(* CoDeSys 2.3.9.41 project: revolution.pro *)
(* Libraries: STANDARD.LIB 4.10.05 10:14:46, IECSFC.LIB 13.4.06 14:51:28, SYSLIBTIME.LIB 20.2.06 13:31:16, SYSTASKINFO.LIB 20.2.06 13:31:38, ANALYZATION.LIB 5.10.99 08:05:06, SYSLIBCALLBACK.LIB 20.2.06 13:31:08, PID_Regulators.lib 28.12.06 17:47:54 *)

(* PLC configuration (modules and I/O channels)
DI0_EKM AT %IX0.0 [BitInput]
DI1_pmp1confirm AT %IX0.1 [BitInput]
DI2_pmp2confirm AT %IX0.2 [BitInput]
DI3_pmp3confirm AT %IX0.3 [BitInput]
DI4_pmp1auto AT %IX0.4 [BitInput]
DI5_pmp2auto AT %IX0.5 [BitInput]
Discrete output 4 bit [ID101] node 1, in %IB1 out %QB1 {PinCount = 4; SafeValueBool = FALSE; SafeValueBool = FALSE; SafeValueBool = FALSE; SafeValueBool = FALSE; Visibility = No}
  DO0_pmp1 AT %QX1.0 [BitOutput]
  DO1_pmp2 AT %QX1.1 [BitOutput]
  DO2_pmp3 AT %QX1.2 [BitOutput]
  DO_alarmLight AT %QX1.3 [BitOutput]
Special output [ID104] node 2, in %IB2 out %QB2 {Visibility = No; PinCount = 1}
  AT %QX2.0 [BitOutput] Special output
AI_pressure AT %ID3.0 [FloatInput] Value
cirTime AT %IW3.1 [WordInput] Circular time
Analog Input [ID107] node 0, in %IB3.0 out %QB3.0
Unifed signal sensor [ID700] node 4, in %IB4 out %QB4 {Type_of_sensor700 = IT_0_20; measure_interval = 0.5; ainlow = 0; ainhigh = 20; first_cor_point = 0; first_delta = 0; second_cor_point = 0; second_delta = 0; third_cor_point = 0; third_delta = 0; Visibility = No}
  AT %ID4.0 [FloatInput] Value
  AT %IW4.1 [WordInput] Circular time
  Analog Input [ID107] node 0, in %IB4.0 out %QB4.0
Unifed signal sensor [ID700] node 5, in %IB5 out %QB5 {Type_of_sensor700 = IT_0_20; measure_interval = 0.5; ainlow = 0; ainhigh = 20; first_cor_point = 0; first_delta = 0; second_cor_point = 0; second_delta = 0; third_cor_point = 0; third_delta = 0; Visibility = No}
  AT %ID5.0 [FloatInput] Value
  AT %IW5.1 [WordInput] Circular time
  Analog Input [ID107] node 0, in %IB5.0 out %QB5.0
Unifed signal sensor [ID700] node 6, in %IB6 out %QB6 {Type_of_sensor700 = IT_0_20; measure_interval = 0.5; ainlow = 0; ainhigh = 20; first_cor_point = 0; first_delta = 0; second_cor_point = 0; second_delta = 0; third_cor_point = 0; third_delta = 0; Visibility = No}
  AT %ID6.0 [FloatInput] Value
  AT %IW6.1 [WordInput] Circular time
  Analog Input [ID107] node 0, in %IB6.0 out %QB6.0
Analog output [ID106] node 7, in %IB7 out %QB7 {DAC_Type = Voltage 0-10 B; Analog_offset_correction = 0; Analog_full_range_correction = 0; SafeValueFloat = 0; Visibility = No}
  AT %QD7.0 [FloatOutput] Value
  AT %QD8.0 [FloatOutput] Value
AT %QD9.0 [DWordOutput] Last address
AT %QW9.1 [WordOutput] Last error
RS-485-1 [COM1_USART] node 0, in %IB9.0 out %QB9.0 {CommunicationSpeed = 19200; Parity = NO PARITY CHECK; BitLength = 8 bits; StopLength = One stop bit; InterfaceType = RS485; FrameOriented = RTU; Timeout = 0; Visibility = No}
AT %QB9.1.0 [ComChannel] Command (0xff - Start)
atv1_freq AT %IW9.1.0.0 [WordInput]
atv1_curr AT %IW9.1.1.0 [WordInput]
atv1_lastError AT %IW9.1.2.0 [WordInput]
atv1_writeHz AT %QW9.1.3.0 [WordOutput]
AT %QB9.2.0 [ComChannel] Command (0xff - Start)
atv2_freq AT %IW9.2.0.0 [WordInput]
atv2_curr AT %IW9.2.1.0 [WordInput]
atv2_lastError AT %IW9.2.2.0 [WordInput]
atv2_writeHz AT %QW9.2.3.0 [WordOutput]
Debug RS-232 [DEBUG_USART] node 0, in %IB10.0.0 out %QB10.0.0 {CommunicationSpeed = 11520; Parity = EVEN; BitLength = 8 bits; StopLength = One stop bit; InterfaceType = RS232; FrameOriented = RTU; Timeout = 0; Visibility = No}
pan_INPUT_ONE AT %QW10.1.0 [WordOutput] setTime
pan_INPUT_TWO AT %QW10.2.0 [WordOutput]
pan_OUTPUT_ONE AT %QW10.3.0 [WordOutput]
pan_OUTPUT_TWO AT %QW10.4.0 [WordOutput]
2 byte [Register] node 5, in %IB10.5 out %QB10.5
  pan_pressure AT %QW10.5.0 [WordOutput]
2 byte [Register] node 6, in %IB10.6 out %QB10.6
  pan_daySetpoint AT %QW10.6.0 [WordOutput]
2 byte [Register] node 7, in %IB10.7 out %QB10.7
  pan_nightSetpoint AT %QW10.7.0 [WordOutput]
2 byte [Register] node 8, in %IB10.8 out %QB10.8
  pan_finishSetpoint AT %QW10.8.0 [WordOutput]
2 byte [Register] node 9, in %IB10.9 out %QB10.9
  pan_pres4ma AT %QW10.9.0 [WordOutput]
2 byte [Register] node 10, in %IB10.10 out %QB10.10
  pan_pres20ma AT %QW10.10.0 [WordOutput]
2 byte [Register] node 11, in %IB10.11 out %QB10.11
  pan_mainPmp AT %QW10.11.0 [WordOutput]
2 byte [Register] node 12, in %IB10.12 out %QB10.12
  pan_resStartDelta AT %QW10.12.0 [WordOutput]
2 byte [Register] node 13, in %IB10.13 out %QB10.13
  pan_resStartDelay AT %QW10.13.0 [WordOutput]
2 byte [Register] node 14, in %IB10.14 out %QB10.14
  pan_resStopHz AT %QW10.14.0 [WordOutput]
2 byte [Register] node 15, in %IB10.15 out %QB10.15
  pan_prop AT %QW10.15.0 [WordOutput]
2 byte [Register] node 16, in %IB10.16 out %QB10.16
  pan_integ AT %QW10.16.0 [WordOutput]
2 byte [Register] node 17, in %IB10.17 out %QB10.17
  pan_diff AT %QW10.17.0 [WordOutput]
2 byte [Register] node 18, in %IB10.18 out %QB10.18
  pan_integMin AT %QW10.18.0 [WordOutput]
2 byte [Register] node 19, in %IB10.19 out %QB10.19
  pan_integMax AT %QW10.19.0 [WordOutput]
2 byte [Register] node 20, in %IB10.20 out %QB10.20
  pan_dryHodDelay AT %QW10.20.0 [WordOutput]
2 byte [Register] node 21, in %IB10.21 out %QB10.21
  pan_aType_1 AT %QW10.21.0 [WordOutput]
2 byte [Register] node 22, in %IB10.22 out %QB10.22
  pan_aType_2 AT %QW10.22.0 [WordOutput]
2 byte [Register] node 23, in %IB10.23 out %QB10.23
  pan_aType_3 AT %QW10.23.0 [WordOutput]
2 byte [Register] node 24, in %IB10.24 out %QB10.24
  pan_aTime_1 AT %QW10.24.0 [WordOutput]
2 byte [Register] node 25, in %IB10.25 out %QB10.25
  pan_aTime_2 AT %QW10.25.0 [WordOutput]
2 byte [Register] node 26, in %IB10.26 out %QB10.26
  pan_aTime_3 AT %QW10.26.0 [WordOutput]
2 byte [Register] node 27, in %IB10.27 out %QB10.27
  pan_aDate_1 AT %QW10.27.0 [WordOutput]
2 byte [Register] node 28, in %IB10.28 out %QB10.28
  pan_aDate_2 AT %QW10.28.0 [WordOutput]
2 byte [Register] node 29, in %IB10.29 out %QB10.29
  pan_aDate_3 AT %QW10.29.0 [WordOutput]
2 byte [Register] node 30, in %IB10.30 out %QB10.30
  pan_aPres_1 AT %QW10.30.0 [WordOutput]
2 byte [Register] node 31, in %IB10.31 out %QB10.31
  pan_aPres_2 AT %QW10.31.0 [WordOutput]
2 byte [Register] node 32, in %IB10.32 out %QB10.32
  pan_aPres_3 AT %QW10.32.0 [WordOutput]
2 byte [Register] node 33, in %IB10.33 out %QB10.33
  pan_aSetpoint_1 AT %QW10.33.0 [WordOutput]
2 byte [Register] node 34, in %IB10.34 out %QB10.34
  pan_aSetpoint_2 AT %QW10.34.0 [WordOutput]
2 byte [Register] node 35, in %IB10.35 out %QB10.35
  pan_aSetpoint_3 AT %QW10.35.0 [WordOutput]
2 byte [Register] node 36, in %IB10.36 out %QB10.36
  pan_aFreq_1 AT %QW10.36.0 [WordOutput]
2 byte [Register] node 37, in %IB10.37 out %QB10.37
  pan_aFreq_2 AT %QW10.37.0 [WordOutput]
2 byte [Register] node 38, in %IB10.38 out %QB10.38
  pan_aFreq_3 AT %QW10.38.0 [WordOutput]
2 byte [Register] node 39, in %IB10.39 out %QB10.39
  pan_aCurr_1 AT %QW10.39.0 [WordOutput]
2 byte [Register] node 40, in %IB10.40 out %QB10.40
  pan_aCurr_2 AT %QW10.40.0 [WordOutput]
2 byte [Register] node 41, in %IB10.41 out %QB10.41
  pan_aCurr_3 AT %QW10.41.0 [WordOutput]
2 byte [Register] node 42, in %IB10.42 out %QB10.42
  pan_aMainPmp_1 AT %QW10.42.0 [WordOutput]
2 byte [Register] node 43, in %IB10.43 out %QB10.43
  pan_aMainPmp_2 AT %QW10.43.0 [WordOutput]
2 byte [Register] node 44, in %IB10.44 out %QB10.44
  pan_aMainPmp_3 AT %QW10.44.0 [WordOutput]
2 byte [Register] node 45, in %IB10.45 out %QB10.45
  pan_topPos AT %QW10.45.0 [WordOutput]
2 byte [Register] node 46, in %IB10.46 out %QB10.46
  pan_midPos AT %QW10.46.0 [WordOutput]
2 byte [Register] node 47, in %IB10.47 out %QB10.47
  pan_bottomPos AT %QW10.47.0 [WordOutput]
2 byte [Register] node 48, in %IB10.48 out %QB10.48
  pan_cursor AT %QW10.48.0 [WordOutput]
2 byte [Register] node 49, in %IB10.49 out %QB10.49
  pan_setHH AT %QW10.49.0 [WordOutput]
2 byte [Register] node 50, in %IB10.50 out %QB10.50
  pan_setMMin AT %QW10.50.0 [WordOutput]
2 byte [Register] node 51, in %IB10.51 out %QB10.51
  pan_setDD AT %QW10.51.0 [WordOutput]
2 byte [Register] node 52, in %IB10.52 out %QB10.52
  pan_setMM AT %QW10.52.0 [WordOutput]
2 byte [Register] node 53, in %IB10.53 out %QB10.53
  pan_setYY AT %QW10.53.0 [WordOutput]
2 byte [Register] node 54, in %IB10.54 out %QB10.54
  pan_currHH AT %QW10.54.0 [WordOutput]
2 byte [Register] node 55, in %IB10.55 out %QB10.55
  pan_currMMin AT %QW10.55.0 [WordOutput]
2 byte [Register] node 56, in %IB10.56 out %QB10.56
  pan_currDD AT %QW10.56.0 [WordOutput]
2 byte [Register] node 57, in %IB10.57 out %QB10.57
  pan_currYY AT %QW10.57.0 [WordOutput]
  pan_ppDelay AT %QW10.58.0 [WordOutput]
  pan_ppLimit AT %QW10.59.0 [WordOutput]
  pan_ppFic AT %QW10.60.0 [WordOutput]
  AT %QW10.61.0 [WordOutput]
  AT %QW10.62.0 [WordOutput]
*)

(* Global variable list: Global_Variables *)
VAR_GLOBAL
	(* Times *)
	GetTime: CurTimeEx;
	TimeAndDate: SystemTimeDate;
	Sys_Time: SysTime64;

	(* Alarms *)
	Alarmy : WORD;

	sensBreak : BOOL; (* 1 *)
	sensShort : BOOL; (* 2 *)
	dryHod		 : BOOL; (* 3 *)
	ekmUpper : BOOL; (* 4 *)
	fcAlarm	: BOOL; (* 5 *)
	kaPmp1fc	: BOOL; (* 6 *)
	kaPmp2fc	: BOOL; (* 7 *)
	kaPmp3fc : BOOL; (* 8 *)
	kaKM1		: BOOL; (* 9 *)
	kaPmp1d : BOOL;  (* 10 *)
	kaPmp2d : BOOL;  (* 11 *)
	kaPmp3d : BOOL;  (* 12 *)
END_VAR

(* POU PLC_PRG, ST *)
PROGRAM PLC_PRG
VAR
	scale : CALIBRATION;
	spcheck : SPDAYCYCLE;
	core : PNS_CORE;
	priority : PRIORITIZATION;
	rotate : ROTATION;
	protect : PRESSURE_PROTECT;

	(* dryHod *)
	dryTimer : TON;
	dryHodOk : BOOL;

	(* Alarmes *)
	breakDetect : BOOL;
	breakTimer : TON;

	shortDetect : BOOL;
	shortTimer : TON;

	fcAlarmDetect, fcAlarmFP : BOOL;
	fcAlarmTimer : TON;

	pmp1kaDetect, pmp2kaDetect, pmp3kaDetect : BOOL;
	pmp1kaDetectD, pmp2kaDetectD, pmp3kaDetectD : BOOL;
	pmp1kaTimer, pmp2kaTimer, pmp3kaTimer : TON;
	pmp1kaTimerD, pmp2kaTimerD, pmp3kaTimerD : TON;
	pmp1kaFP, pmp2kaFP, pmp3kaFP,  kmKaFP : BOOL;
	pmp1kaFPD, pmp2kaFPD, pmp3kaFPD,  kmKaFPD : BOOL;
	fc_state, fc_kaDetect : BOOL;
	fcKaTimer : TON;

	(* Times *)
	setTime : BOOL;
END_VAR
VAR RETAIN
	(* dry hod *)
	dryDelay : TIME;

	(* Pressure *)
	daySetpoint, nightSetpoint : REAL;

	(*Calibration *)
	pres4ma, pres20ma : REAL;

	(* Process *)
	resStartDelta : REAL;
	resStartDelay : TIME;
	resStopHz : WORD;

	(* PID *)
	prop : REAL;
	integ : DINT;

	(* Pressure Protect *)
	ppDelay : TIME;
	ppLimit : REAL;
	ppFic : REAL;

END_VAR
dryTimer(IN:= DI0_EKM, PT:=dryDelay, Q=>dryHodOk, ET=> );

Inputs;



Times;
END_PROGRAM
ACTION Alarmes:
(* SENS BREAK *)
IF AI_pressure < 3.8 THEN
	breakDetect := TRUE;
ELSE
	breakDetect := FALSE;
END_IF;

breakTimer(IN:= breakDetect, PT:=T#1s, Q=>sensBreak, ET=> );


(* SENS SHORT *)
IF AI_pressure > 21.0 THEN
	shortDetect := TRUE;
ELSE
	shortDetect := FALSE;
END_IF;

shortTimer(IN:= shortDetect, PT:=T#1s, Q=>sensShort, ET=> );

(* DRY HOD *)
dryHod := dryHodOk;

(* EKM UPPER *)

(* FC ALARM *)
(*
IF DI_fcAlarm AND fc_on = TRUE THEN
	fcAlarmDetect := TRUE;
ELSE
	fcAlarmDetect := FALSE;
END_IF;

fcAlarmTimer(IN:= fcAlarmDetect, PT:=T#10s, Q=>fcAlarm, ET=> );

IF fcAlarm AND fcAlarmFP = FALSE THEN
	fcAlarmFP := TRUE;
	ShiftKtpMainPmp;
END_IF;

IF fcAlarm = FALSE THEN
	fcAlarmFP := FALSE;
END_IF;
*)
(* PMP1 KA *)
	(* FC *)
(*
IF pmp1fc AND pmp1_state = FALSE THEN
	pmp1kaDetect := TRUE;
ELSE
	pmp1kaDetect := FALSE;
END_IF;
	(* Direct *)
IF pmp1d AND pmp1_stateD = FALSE THEN
	pmp1kaDetectD := TRUE;
ELSE
	pmp1kaDetectD := FALSE;
END_IF;
*)
(*
pmp1kaTimer(IN:= pmp1kaDetect, PT:=T#10s, Q=>kaPmp1fc, ET=> );
pmp1kaTimerD(IN:= pmp1kaDetectD, PT:=T#10s, Q=>kaPmp1d, ET=> );
*)
(*
(* FC *)
IF kaPmp1fc AND pmp1kaFP = FALSE THEN
	pmp1kaFP := TRUE;
	pmp1kaSave := TRUE;
	ShiftKtpMainPmp;
END_IF;

IF kaPmp1fc = FALSE THEN
	pmp1kaFP := FALSE;
END_IF;
(* Direct *)
IF kaPmp1d AND pmp1kaFPD = FALSE THEN
	pmp1kaFPD := TRUE;
	pmp1kaSaveD := TRUE;
END_IF;

IF kaPmp1d = FALSE THEN
	pmp1kaFPD := FALSE;
END_IF;
*)
(*
(* PMP2 KA *)
IF pmp2fc AND pmp2_state = FALSE THEN
	pmp2kaDetect := TRUE;
ELSE
	pmp2kaDetect := FALSE;
END_IF;

IF pmp2d AND pmp2_stateD = FALSE THEN
	pmp2kaDetectD := TRUE;
ELSE
	pmp2kaDetectD := FALSE;
END_IF;

pmp2kaTimer(IN:= pmp2kaDetect, PT:=T#10s, Q=>kaPmp2fc, ET=> );
pmp2kaTimerD(IN:= pmp2kaDetectD, PT:=T#10s, Q=>kaPmp2d, ET=> );

IF kaPmp2fc AND pmp2kaFP = FALSE THEN
	pmp2kaFP := TRUE;
	pmp2kaSave := TRUE;
END_IF;

IF kaPmp2fc = FALSE THEN
	pmp2kaFP := FALSE;
END_IF;

IF kaPmp2d AND pmp2kaFPD = FALSE THEN
	pmp2kaFPD := TRUE;
	pmp2kaSaveD := TRUE;
END_IF;

IF kaPmp2d = FALSE THEN
	pmp2kaFPD := FALSE;
END_IF;

(* PMP3 KA *)
IF pmp3fc AND pmp3_state = FALSE THEN
	pmp3kaDetect := TRUE;
ELSE
	pmp3kaDetect := FALSE;
END_IF;

IF pmp3d AND pmp3_stateD = FALSE THEN
	pmp3kaDetectD := TRUE;
ELSE
	pmp3kaDetectD := FALSE;
END_IF;

pmp3kaTimer(IN:= pmp3kaDetect, PT:=T#10s, Q=>kaPmp3fc, ET=> );
pmp3kaTimerD(IN:= pmp3kaDetectD, PT:=T#10s, Q=>kaPmp3d, ET=> );

IF kaPmp3fc AND pmp3kaFP = FALSE THEN
	pmp3kaFP := TRUE;
	pmp3kaSave := TRUE;
	ShiftKtpMainPmp;
END_IF;

IF kaPmp3fc = FALSE THEN
	pmp3kaFP := FALSE;
END_IF;

IF kaPmp3d AND pmp3kaFPD = FALSE THEN
	pmp3kaFPD := TRUE;
	pmp3kaSaveD := TRUE;
END_IF;

IF kaPmp3d = FALSE THEN
	pmp3kaFPD := FALSE;
END_IF;

IF ktp_INPUT.1 THEN
	pmp1kaSave := FALSE;
	pmp2kaSave := FALSE;
	pmp3kaSave := FALSE;
	pmp1kaSaveD := FALSE;
	pmp2kaSaveD := FALSE;
	pmp3kaSaveD := FALSE;
	ktp_INPUT.1 := FALSE;
END_IF;

(* FC KA *)
IF fc_on AND fc_state = FALSE THEN
	fc_kaDetect := TRUE;
ELSE
	fc_kaDetect := FALSE;
END_IF;

fcKaTimer(IN:= fc_kaDetect, PT:=T#10s, Q=>kaKM1, ET=> );

IF kaKM1 AND kmKaFP = FALSE THEN
	kmKaFP := TRUE;
	ShiftKtpMainPmp;
END_IF;

IF kaKM1 = FALSE THEN
	kmKaFP := FALSE;
END_IF;

(* ALARMY *)
Alarmy.0 := sensBreak;
Alarmy.1 := sensShort;
Alarmy.2 := dryHod;

Alarmy.4 := fcAlarm;
Alarmy.5 := kaPmp1fc;
Alarmy.6 := kaPmp2fc;
Alarmy.7 := kaPmp3fc;
Alarmy.8 := kaKM1;

IF Alarmy > 0 THEN
	DO_lamp_fcAlarm := TRUE;
ELSE
	DO_lamp_fcAlarm := FALSE;
END_IF;
*)
END_ACTION
ACTION Inputs:
setTime := pan_INPUT_ONE.0;

drydelay := WORD_TO_TIME ( pan_dryHoddelay * 1000 );

daySetpoint := WORD_TO_REAL ( pan_daySetpoint ) / 100;
nightSetpoint := WORD_TO_REAL ( pan_nightSetpoint ) / 100;

pres4ma := WORD_TO_REAL ( pan_pres4ma ) / 100;
pres20ma := WORD_TO_REAL ( pan_pres20ma ) / 100;

resStartDelta := WORD_TO_REAL ( pan_resStartDelta ) / 100;
resStartDelay := WORD_TO_TIME ( pan_resStartDelay * 1000 );
resStopHz := resStopHz;

prop := WORD_TO_REAL ( pan_prop ) / 100;
integ := pan_integ;

ppDelay := WORD_TO_TIME ( pan_ppDelay * 1000 );
ppLimit := WORD_TO_REAL ( pan_ppLimit ) / 100;
ppFic := WORD_TO_REAL ( pan_ppFic ) / 100;
END_ACTION
ACTION Times:
TimeAndDate.Day :=0;
TimeAndDate.DayOfWeek :=0;
TimeAndDate.dwHighMsec :=0;
TimeAndDate.dwLowMSecs :=0;
TimeAndDate.Milliseconds :=0;
TimeAndDate.Minute :=0;
TimeAndDate.Second :=0;
TimeAndDate.Hour :=0;
TimeAndDate.Year :=0;
TimeAndDate.Month :=0;
Sys_time.ulHigh :=0;
Sys_time.ulLow :=0;
GetTime (SystemTime:=Sys_Time , TimeDate:= TimeAndDate);


IF pan_INPUT_ONE.0 THEN
	TimeAndDate.Minute:=pan_setMMin;
	TimeAndDate.Second:=10;
	TimeAndDate.Hour:=pan_setHH;
	TimeAndDate.Day:=pan_setDD;
	TimeAndDate.Month:=pan_setMM;
	TimeAndDate.Year:=pan_setYY;
	GetTime (SystemTime:=Sys_Time , TimeDate:= TimeAndDate);

	pan_INPUT_ONE.0 := FALSE;
END_IF;
END_ACTION

(* POU CALIBRATION, ST *)
FUNCTION_BLOCK CALIBRATION
VAR_INPUT
	AI_RAW : REAL;
	r_bar4ma : REAL;
	w2d_bar4ma : WORD;
	r_bar20ma : REAL;
	w2d_bar20ma : WORD;
END_VAR
VAR_OUTPUT
	r_scaled : REAL;
	w2d_scaled : WORD;
END_VAR
VAR
END_VAR
(* Result = n2 + ( Input - n1 ) * ( ( m2 - n2 ) / ( m1 - n1 ) ) *)

w2d_scaled := w2d_bar4ma  + ( REAL_TO_INT( AI_RAW * 100 ) - 400 ) * ( w2d_bar20ma - w2d_bar4ma ) / 1600;

r_scaled := r_bar4ma  + ( AI_RAW - 4.0 ) * ( r_bar20ma - r_bar4ma ) / 16;
END_FUNCTION_BLOCK

(* POU SPDAYCYCLE, ST *)
FUNCTION_BLOCK SPDAYCYCLE
VAR_INPUT
	firstSetpoint : REAL;
	secondSetpoint : REAL;
	spHHfirst : WORD;
	spMMfirst : WORD;
	spHHsecond : WORD;
	spMMsecond : WORD;
	HH, MM : WORD;
END_VAR
VAR_OUTPUT
	setpoint : REAL;
END_VAR
VAR
END_VAR
IF spHHsecond > spHHfirst THEN
	IF HH = spHHsecond AND MM >= spMMsecond THEN
		setpoint := secondSetpoint;
	END_IF;
	IF HH > spHHsecond AND HH > spHHfirst THEN
		setpoint := secondSetpoint;
	END_IF;
	IF HH >= 0 AND HH < spHHfirst THEN
		setpoint := secondSetpoint;
	END_IF;
	IF HH = spHHfirst AND MM < spMMfirst THEN
		setpoint := secondSetpoint;
	END_IF;
	IF HH = spHHfirst AND MM >= spMMfirst THEN
		setpoint := firstSetpoint;
	END_IF;
	IF HH > spHHfirst AND HH < spHHsecond THEN
		setpoint := firstSetpoint;
	END_IF;
	IF HH = spHHsecond AND MM < spMMsecond THEN
		setpoint := firstSetpoint;
	END_IF;
END_IF;

IF spHHsecond < spHHfirst THEN
	IF HH = spHHsecond AND MM >= spMMsecond THEN
		setpoint := secondSetpoint;
	END_IF;
	IF HH > spHHsecond AND HH < spHHfirst THEN
		setpoint := secondSetpoint;
	END_IF;
	IF HH = spHHfirst AND MM < spMMfirst THEN
		setpoint := secondSetpoint;
	END_IF;
	IF HH = spHHfirst AND MM >= spMMfirst THEN
		setpoint := firstSetpoint;
	END_IF;
	IF HH > spHHfirst THEN
		setpoint := firstSetpoint;
	END_IF;
	IF HH >= 0 AND spHHsecond > 0 THEN
		setpoint := firstSetpoint;
	END_IF;
	IF HH = spHHsecond AND MM < spMMsecond THEN
		setpoint := firstSetpoint;
	END_IF;
END_IF;
END_FUNCTION_BLOCK

(* POU PNS_CORE, ST *)
FUNCTION_BLOCK PNS_CORE
VAR_INPUT
	FAULT : BOOL;
	pressure : REAL;
	setpoint : REAL;
	resStart_hz : REAL;
	resStart_delta : REAL;
	resStart_delay : TIME;
	resStop_hz : REAL;
	resStop_delay : TIME;
	pid_prop : REAL;
	pid_integ : DINT;

END_VAR
VAR_OUTPUT
	main : BOOL;
	reserve : BOOL;
	secRes : BOOL;
	hz : REAL;
END_VAR
VAR
	(* PID *)
	pid : PID_FUNCTION;
	real_pres, real_setpoint, pid_out : REAL;
	prop : REAL;
	diff : REAL;
	integ : DINT;
	integMin, integMax : REAL;
	(* Process *)
	resStartTimerGo : BOOL;
	resStartTimer : TON;
	resAllowedByConditions : BOOL;
	resStopTimerGo : BOOL;
	resStopTimer : TON;
	resStoppedByConditions : BOOL;
END_VAR
PID;

IF FAULT = FALSE THEN
	main := TRUE;
END_IF;

(* включение резервного *)
IF ( resStart_hz < hz ) AND ( resStart_delta < setpoint - pressure ) THEN
	resStartTimerGo := TRUE;
ELSE
	resStartTimerGo := FALSE;
END_IF;

resStartTimer(IN:= resStartTimerGo, PT:=resStart_delay, Q=>resAllowedByConditions, ET=> );

IF resAllowedByConditions THEN
	reserve := TRUE;
END_IF;

(* выключение резервного *)
IF ( resStop_hz > hz ) THEN
	resStopTimerGo := TRUE;
ELSE
	resStopTimerGo := FALSE;
END_IF;

resStartTimer(IN:= resStopTimerGo, PT:=resStop_delay, Q=>resStoppedByConditions, ET=> );

IF ( resStoppedByConditions ) THEN
	reserve := FALSE;
END_IF;

IF FAULT = TRUE THEN
	main := FALSE;
	reserve := FALSE;
	secRes := FALSE;
END_IF;
END_FUNCTION_BLOCK
ACTION PID:
pid(
			PV:= pressure, (* REAL Входное значение*)
			PV_TIME:= cirTime, (* WORD Время получения входной величины - отсчитвыается в долях секунды и берется из UNIVERSAL Sensor/ Circular time*)
			SP:= setpoint, (* REAL уставка*)
			PB:= prop, (*REAL полоса пропорциональности*)
			TI_:= integ, (* DINT постоянная интегрирования - 4 байтовое целое знаковое*)
			TD_:= diff, (* REAL постоянная диффереренцирования*)
			_IMIN:= -1.0, (* REAL минимум интегральной составляющей*)
			_IMAX:= 1.0, (* REAL максимум интегральной составляющей*)
			OUT_VAL=> hz); (* REAL Выходное значение*)
END_ACTION

(* POU PRIORITIZATION, ST *)
FUNCTION_BLOCK PRIORITIZATION
VAR_INPUT
	mainPmp_N_in : INT;
	mainMustStart : BOOL;
	resMustStart : BOOL;
	(*secRes : BOOL;*)
	pmp1auto : BOOL;
	pmp2auto : BOOL;
	(*pmp3auto : BOOL;*)
	pmp1fault : BOOL;
	pmp2fault : BOOL;
END_VAR
VAR_OUTPUT
	mainPmp_N_out : INT;
	pmp1start : BOOL;
	pmp2start : BOOL;
	(*pmp3start : BOOL;*)
END_VAR
VAR
	pmp1ready : BOOL;
	pmp2ready : BOOL;
	pmp1priority : INT;
	pmp2priority : INT;
	shiftMain : SHIFT;
END_VAR
mainPmp_N_out := mainPmp_N_in;
pmp1priority := 0;
pmp2priority := 0;

CheckMain;

CheckReserve;

pmp1start := FALSE;
pmp2start := FALSE;

IF mainMustStart THEN
	IF pmp1priority = 1 THEN
		pmp1start := TRUE;
	END_IF;
	IF pmp2priority = 1 THEN
		pmp2start := TRUE;
	END_IF;
END_IF;

IF resMustStart THEN
	IF pmp1priority = 2 THEN
		pmp1start := TRUE;
	END_IF;
	IF pmp2priority = 2 THEN
		pmp2start := TRUE;
	END_IF;
END_IF;
END_FUNCTION_BLOCK
ACTION CheckMain:
IF ( pmp1auto = TRUE ) AND ( pmp1fault = FALSE ) THEN
	pmp1ready := TRUE;
ELSE
	pmp1ready := FALSE;
END_IF;

IF ( pmp2auto = TRUE ) AND ( pmp2fault = FALSE ) THEN
	pmp2ready := TRUE;
ELSE
	pmp2ready := FALSE;
END_IF;

IF NOT pmp1ready  AND NOT pmp2ready THEN
	mainPmp_N_out := 0;
END_IF;

IF mainPmp_N_out = 1 THEN
	IF NOT pmp1ready THEN
		shiftMain( mainPmp_N_in := mainPmp_N_out, pumpCount := 2, mainPmp_N_out => mainPmp_N_out);
	END_IF;
END_IF;

IF mainPmp_N_out = 2 THEN
	IF NOT pmp2ready THEN
		shiftMain( mainPmp_N_in := mainPmp_N_out, pumpCount := 2, mainPmp_N_out => mainPmp_N_out);
	END_IF;
END_IF;

IF mainPmp_N_out = 0 THEN
	IF pmp1ready THEN
		mainPmp_N_out := 1;
	ELSE
		IF pmp2ready THEN
			mainPmp_N_out := 2;
		END_IF;
	END_IF;
END_IF;

IF mainPmp_N_out = 1 THEN
	pmp1priority := 1;
END_IF;

IF mainPmp_N_out = 2 THEN
	pmp2priority := 1;
END_IF;

IF NOT pmp1ready THEN
	pmp1priority := 0;
END_IF;

IF NOT pmp2ready THEN
	pmp2priority := 0;
END_IF;

IF mainPmp_N_out = 0 THEN
	pmp1priority := 0;
	pmp2priority := 0;
END_IF;
END_ACTION
ACTION CheckReserve:
IF pmp1priority = 1 THEN
	IF pmp2ready THEN
		pmp2priority := 2;
	ELSE
		pmp2priority := 0;
	END_IF;
END_IF;

IF pmp2priority = 1 THEN
	IF pmp1ready THEN
		pmp1priority := 2;
	ELSE
		pmp1priority := 0;
	END_IF;
END_IF;
END_ACTION
ACTION ShiftMain:
mainPmp_N_out := mainPmp_N_in + 1;

IF mainPmp_N_out > 2 OR mainPmp_N_out = 0 THEN
	mainPmp_N_out := 1;
END_IF;
END_ACTION

(* POU SHIFT, ST *)
FUNCTION_BLOCK SHIFT
VAR_INPUT
	mainPmp_N_in : INT;
	pumpCount : INT;
END_VAR
VAR_OUTPUT
	mainPmp_N_out : INT;
END_VAR
VAR
	tempMainOut : INT;
END_VAR
tempMainOut := mainPmp_N_in + 1;

IF tempMainOut > pumpCount OR tempMainOut = 0 THEN
	tempMainOut := 1;
END_IF;

mainPmp_N_out := tempMainOut;
END_FUNCTION_BLOCK

(* POU ROTATION, ST *)
FUNCTION_BLOCK ROTATION
VAR_INPUT
	mainPmp_N_in : INT;
	WEEKDAYS : WORD;
	HH : WORD;
	MM : WORD;
END_VAR
VAR_OUTPUT
	mainPmp_N_out : INT;
END_VAR
VAR
	rotateShift : SHIFT;
	rotate : BOOL;
	saveMM : WORD;
END_VAR
rotate := FALSE;

IF ( TimeAndDate.Hour = HH ) AND ( TimeAndDate.Minute = MM ) AND ( saveMM <> MM ) THEN
	CASE TimeAndDate.DayOfWeek OF
		1 : IF WEEKDAYS.0 THEN rotate := TRUE; END_IF;
		2 : IF WEEKDAYS.1 THEN rotate := TRUE; END_IF;
		3 : IF WEEKDAYS.3 THEN rotate := TRUE; END_IF;
		4 : IF WEEKDAYS.4 THEN rotate := TRUE; END_IF;
		5 : IF WEEKDAYS.5 THEN rotate := TRUE; END_IF;
		6 : IF WEEKDAYS.6 THEN rotate := TRUE; END_IF;
		7 : IF WEEKDAYS.6 THEN rotate := TRUE; END_IF;
	END_CASE;
ELSE
	saveMM := 70;
END_IF;

IF rotate THEN
	rotateShift( mainPmp_N_in := mainPmp_N_in, pumpCount := 2, mainPmp_N_out => mainPmp_N_out );
	saveMM := MM;
	rotate := FALSE;
END_IF;
END_FUNCTION_BLOCK

(* POU PRESSURE_PROTECT, ST *)
FUNCTION_BLOCK PRESSURE_PROTECT
VAR_INPUT
	(*hz : REAL;*)
	pressure : REAL;
	setpoint_in : REAL;
	(*protectFactor : REAL;*)
	delay : TIME;
	limitPres : REAL;
	ficSetpoint : REAL;
END_VAR
VAR_OUTPUT
	setpoint_out : REAL;
END_VAR
VAR
	protectActive : BOOL;
	overpressure : BOOL;
	(*delta : REAL;*)
	(*ratio : REAL;*)
	overpresTimer : TON;
	(*excessConfirmed : BOOL;*)
	(*predelay : REAL;*)
END_VAR
protectActive := FALSE;

IF pressure > limitPres THEN
	overpressure := TRUE;
ELSE
	overpressure := FALSE;
END_IF;

overpresTimer(IN:= overpressure, PT:= delay );

IF overpresTimer.Q THEN
	protectActive := TRUE;
END_IF;

IF protectActive AND ( pressure < setpoint_in ) THEN
	protectActive := FALSE;
END_IF;

IF protectActive THEN
	setpoint_out := ficSetpoint;
ELSE
	setpoint_out := setpoint_in;
END_IF;

(* BULLSHIT
setpoint_out := setpoint_in;

delta := pressure - setpoint_in;
ratio := pressure / setpoint_in;

IF delta > 0 THEN
	overpressure := TRUE;
ELSE
	overpressure := FALSE;
END_IF;

predelay := 100 - EXPT(1.1, delta*protectFactor);
IF predelay < 0 THEN predelay := 1; END_IF;
delay := REAL_TO_TIME ( predelay * 1000)

overpresTimer(IN:= overpressure, PT:= delay, Q=> excessConfirmed, ET=> );

IF excessConfirmed THEN
	setpoint_out := setpoint_in / ratio;
END_IF;
/BULLSHIT *)
END_FUNCTION_BLOCK

(* POU ALARMS, ST *)
PROGRAM ALARMS
VAR
	fp_sensBreak : BOOL; (* 1 *)
	fp_sensShort  : BOOL; (* 2 *)
	fp_ekmLower  : BOOL; (* 3 *)
	fp_ekmUpper  : BOOL; (* 4 *)
	fp_fcAlarm		 : BOOL; (* 5 *)
	fp_kaPmp1fc	 : BOOL; (* 6 *)
	fp_kaPmp2fc	 : BOOL; (* 7 *)
	fp_kaPmp3fc 	 : BOOL; (* 8 *)
	fp_kaKM1		 : BOOL; (* 9 *)
	aPowerOffFP 	: BOOL; (* 10 *)
	fp_kaPmp1d	 : BOOL; (* 11 *)
	fp_kaPmp2d	 : BOOL; (* 12 *)
	fp_kaPmp3d 	 : BOOL; (* 13 *)
	last_aType 	:  WORD;

	topPos, midPos, bottomPos : INT;


END_VAR
VAR RETAIN
	id	: INT;
	(* must be retain *)
	aType 		: ARRAY[0..99] OF WORD;
	aTime 		: ARRAY[0..99] OF WORD;
	aDate 		: ARRAY[0..99] OF WORD;
	pres		: ARRAY[0..99] OF WORD;
	setpoint	: ARRAY[0..99] OF WORD;
	freq		: ARRAY[0..99] OF WORD;
	curr		: ARRAY[0..99] OF WORD;
	mainPmp 	: ARRAY[0..99] OF WORD;

END_VAR
last_aType := 0;

IF pan_cursor = 127 THEN
	PutCursorToLastAlarm;
END_IF

CorrectCursor;

FillFields;

Check;

pan_topPos := INT_TO_WORD( topPos );
pan_midPos := INT_TO_WORD( midPos );
pan_bottomPos := INT_TO_WORD( bottomPos );
END_PROGRAM
ACTION AddNew:
aType[ id ] := last_aType;
aTime[ id ] := TimeAndDate.Hour * 100 + TimeAndDate.Minute;
aDate[ id ] := TimeAndDate.Day * 100 + TimeAndDate.Month;
pres[ id ] := pan_pressure;
setpoint[ id ] := pan_finishSetpoint;
freq[ id ] := 0;
curr[ id ] := 0;
mainPmp[ id ] := pan_mainPmp;

id := id + 1;

IF id >= 100 THEN
	id := 0;
END_IF;

pan_cursor := INT_TO_WORD( id );
END_ACTION
ACTION Check:
(* SENS BREAK *)
IF sensBreak AND fp_sensBreak = FALSE THEN
	fp_sensBreak := TRUE;
	last_aType := 1;
	AddNew;
END_IF;

IF sensBreak = FALSE THEN
	fp_sensBreak := FALSE;
END_IF;

(* SENS SHORT *)
IF sensShort AND fp_sensShort = FALSE THEN
	fp_sensShort := TRUE;
	last_aType := 2;
	AddNew;
END_IF;

IF sensShort = FALSE THEN
	fp_sensShort := FALSE;
END_IF;

(* EKM LOWER *)
IF dryHod AND fp_ekmLower = FALSE THEN
	fp_ekmLower := TRUE;
	last_aType := 3;
	AddNew;
END_IF;

IF dryHod = FALSE THEN
	fp_ekmLower := FALSE;
END_IF;

(* EKM UPPER *)
IF ekmUpper AND fp_ekmUpper = FALSE THEN
	fp_ekmUpper := TRUE;
	last_aType := 4;
	AddNew;
END_IF;

IF ekmUpper = FALSE THEN
	fp_ekmUpper := FALSE;
END_IF;

(* FC ALARM *)
IF fcAlarm AND fp_fcAlarm = FALSE THEN
	fp_fcAlarm := TRUE;
	last_aType := 5;
	AddNew;
END_IF;

IF fcAlarm = FALSE THEN
	fp_fcAlarm := FALSE;
END_IF;

(* KA PMP1FC *)
IF kaPmp1fc AND fp_kaPmp1fc = FALSE THEN
	fp_kaPmp1fc := TRUE;
	last_aType := 6;
	AddNew;
END_IF;

IF kaPmp1fc = FALSE THEN
	fp_kaPmp1fc := FALSE;
END_IF;

(* KA PMP2FC *)
IF kaPmp2fc AND fp_kaPmp2fc = FALSE THEN
	fp_kaPmp2fc := TRUE;
	last_aType := 7;
	AddNew;
END_IF;

IF kaPmp2fc = FALSE THEN
	fp_kaPmp2fc := FALSE;
END_IF;

(* KA PMP3FC *)
IF kaPmp3fc AND fp_kaPmp3fc = FALSE THEN
	fp_kaPmp3fc := TRUE;
	last_aType := 8;
	AddNew;
END_IF;

IF kaPmp3fc = FALSE THEN
	fp_kaPmp3fc := FALSE;
END_IF;


(* KA PMP1D *)
IF kaPmp1d AND fp_kaPmp1fc = FALSE THEN
	fp_kaPmp1d := TRUE;
	last_aType := 12;
	AddNew;
END_IF;

IF kaPmp1d = FALSE THEN
	fp_kaPmp1d := FALSE;
END_IF;

(* KA PMP2D *)
IF kaPmp2d AND fp_kaPmp2d = FALSE THEN
	fp_kaPmp2d := TRUE;
	last_aType := 13;
	AddNew;
END_IF;

IF kaPmp2d = FALSE THEN
	fp_kaPmp2d := FALSE;
END_IF;

(* KA PMP3D *)
IF kaPmp3d AND fp_kaPmp3d = FALSE THEN
	fp_kaPmp3d := TRUE;
	last_aType := 14;
	AddNew;
END_IF;

IF kaPmp3d = FALSE THEN
	fp_kaPmp3d := FALSE;
END_IF;


(* KA KM1 *)
IF kaKM1 AND fp_kaKM1 = FALSE THEN
	fp_kaKM1 := TRUE;
	last_aType := 9;
	AddNew;
END_IF;

IF kaKM1 = FALSE THEN
	fp_kaKM1 := FALSE;
END_IF;

(* POWER *)
(*
IF powerStatus = FALSE AND aPowerOffFP = FALSE  THEN
	aPowerOffFP := TRUE;
	last_aType := 10;
	AddNew;
END_IF;

IF powerStatus THEN
	aPowerOffFP := FALSE;
END_IF;
*)
END_ACTION
ACTION CorrectCursor:
IF pan_cursor > 99 THEN
	pan_cursor := 0;
END_IF;

topPos := pan_cursor;

midPos := pan_cursor - 1;

bottomPos := pan_cursor - 2;

IF pan_cursor = 0 THEN
	midPos := 99;
	bottomPos := 98;
END_IF;

IF pan_cursor = 1 THEN
	bottomPos := 99;
END_IF;
END_ACTION
ACTION FillFields:
pan_aType_1 		:= aType		[ topPos ];
pan_aTime_1 		:= aTime		[ topPos ];
pan_aDate_1 		:= aDate		[ topPos ];
pan_aPres_1 		:= pres			[ topPos ];
pan_aSetpoint_1	 := setpoint	[ topPos ];
pan_aFreq_1 		:= freq			[ topPos ];
pan_aCurr_1	 	:= curr			[ topPos ];
pan_aMainPmp_1 := mainPmp	[ topPos ];

pan_aType_2 		:= aType		[ midPos ];
pan_aTime_2 		:= aTime		[ midPos ];
pan_aDate_2		:= aDate		[ midPos ];
pan_aPres_2 		:= pres			[ midPos ];
pan_aSetpoint_2 	:= setpoint		[ midPos ];
pan_aFreq_2 		:= freq			[ midPos ];
pan_aCurr_2 		:= curr			[ midPos ];
pan_aMainPmp_2 := mainPmp	[ midPos ];

pan_aType_3 		:= aType		[ bottomPos ];
pan_aTime_3 		:= aTime		[ bottomPos ];
pan_aDate_3		:= aDate		[ bottomPos ];
pan_aPres_3 		:= pres			[ bottomPos ];
pan_aSetpoint_3 	:= setpoint		[ bottomPos ];
pan_aFreq_3 		:= freq			[ bottomPos ];
pan_aCurr_3 		:= curr			[ bottomPos ];
pan_aMainPmp_3 := mainPmp	[ bottomPos ];
END_ACTION
ACTION PutCursorToLastAlarm:
pan_cursor := INT_TO_WORD( id ) - 1;
END_ACTION
